# B&R Automation Studio project condmon
Automation Studio 4.6.3.55 SP

## Configuration X20CP3585

CPU X20CP3585, AutomationRuntime B4.62, Build 4.1.2, Safety 0.0, Vc 

### Task classes (Cpu.sw)
```
Cyclic#1 (cycle 1000 us, tolerance 1000 us):
  rdbuf <- rdbuf.prg
Binaries: udbdef, FWRules, TCData, iomap, ashwac, Role, sysconf, arconfig, asfw, User, ashwd, vccdt, vccbmp, Visu03, vccline, vcfile, arial, vctcal, vcrt, vcmgr, arsvcreg, vccstr, vcbclass, vccbtn, vcgclass, vcdsint, vcnet, vcchtml, Visu01, Visu, vcshared, vcclbox, vccddbox, vccscale, arialbd, vcxml, vccnum, vcpdvnc, vccalarm, vccurl, vccslider, vccbar, vcctext, vccpiech, vcpdsw, vcfntttf, vccovl, vccshape, vcalarm, vcpkat, Visu02, vcctrend, vccpopup, vcdsloc, vcchspot, vcpfx20, Config, Config_2, Config_1
Libraries: operator, runtime, astime, AsIecCon, AsIOVib, AsFltGen, brsystem, sys_lib, DataObj, asstring, standard, vcresman, asbrstr, ashw, MpAlarmX, MpFile, MpBase, AsSem, MpWebXs
```

### Hardware
```
X20BM31 : X20BM31 v1.0.0.1  [X2X1 -> X20CP3585.IF6]
X20CM4810 : X20CM4810 v1.4.4.0  [SS1 -> X20TB12.SS; SL -> X20BM31.SL1]
  Supervision = off
  Current01 = on
  FrequencyBandEnable01 = off
  FrequencyBandEnable02 = off
  FrequencyBandEnable03 = off
  FrequencyBandEnable09 = off
  FrequencyBandEnable10 = off
  FrequencyBandEnable11 = off
  FrequencyBandEnable17 = off
  FrequencyBandEnable18 = off
  FrequencyBandEnable19 = off
  FrequencyBandEnable25 = off
  FrequencyBandEnable26 = off
  FrequencyBandEnable27 = off
X20CP3585 : X20CP3585 v1.5.0.0
  Connector IF2:
    ActivateDevice = 1
    HostName = conmon
    Mode = Manual
    InternetAddress = 192.168.0.34
    SubnetMask = 255.255.255.0
  Connector IF6:
    CycleTime = 1000
    Stations = 16
    AsyncPayload = 160
    OutputJustInTime = off
  ConfigurationID = firstStart_X20CP3585
  Cyclic1Duration = 1000
  Cyclic1Tolerance = 1000
  FileDevice1
  FileDeviceName1 = HD
  FileDevicePath1 = F:\
  FtpUser1
  FtpUsername1 = user
  FtpUserPassword1 = IKmmIU0UA42VIUZbb7SMTTmDelvdeU0oRhYqfrVB1tM=
  FtpUserSalt1 = 73ZO5cbR
  FTPAccessRight1 = 0
X20TB12 : X20TB12 v1.0.0.0
```

### IoMap.iom - X20CP3585/IoMap.iom
```iecst
VAR_CONFIG
	::rdbuf:fb.ioMapping.RequestBufferLock01 AT %QX."X20CM4810".RequestBufferLock01;
	::rdbuf:fb.ioMapping.BufferLockValid01 AT %IX."X20CM4810".BufferLockValid01;
	::rdbuf:fb.ioMapping.BufferInputSequence01 AT %IB."X20CM4810".BufferInputSequence01;
	::rdbuf:fb.ioMapping.BufferRxByte01 AT %IB."X20CM4810".BufferRxByte01;
	::rdbuf:fb.ioMapping.BufferRxByte02 AT %IB."X20CM4810".BufferRxByte02;
	::rdbuf:fb.ioMapping.BufferRxByte03 AT %IB."X20CM4810".BufferRxByte03;
	::rdbuf:fb.ioMapping.BufferRxByte04 AT %IB."X20CM4810".BufferRxByte04;
	::rdbuf:fb.ioMapping.BufferRxByte05 AT %IB."X20CM4810".BufferRxByte05;
	::rdbuf:fb.ioMapping.BufferOutputSequence01 AT %QB."X20CM4810".BufferOutputSequence01;
	::rdbuf:fb.ioMapping.BufferTxByte01 AT %QB."X20CM4810".BufferTxByte01;
	::rdbuf:fb.ioMapping.BufferTxByte02 AT %QB."X20CM4810".BufferTxByte02;
	::rdbuf:fb.ioMapping.BufferTxByte03 AT %QB."X20CM4810".BufferTxByte03;
	::rdbuf:fb.ioMapping.BufferTxByte03 AT %QB."X20CM4810".BufferTxByte04;
END_VAR
```

## Logical view

Binary libraries used (declarations not repeated): operator, runtime, astime, AsIecCon, AsIOVib, AsFltGen, brsystem, sys_lib, DataObj, asstring, standard

### Global.typ - Globale Datentypen
```iecst
TYPE
	CM4810_Data : 	STRUCT
		xAxis : ARRAY[0..8191]OF REAL;
		yAxis : ARRAY[0..8191]OF REAL;
	END_STRUCT;
END_TYPE
```


### Program Logical/rdbuf (IEC)

#### Variables.var
```iecst
VAR
	fb : vbioCtrlCM4810Ex1;
	bufferUploadDuration : TIME;
	cmdUploadBuffer : USINT;
	cycleCounter : UDINT;
	step : UINT;
	rtinfo : RTInfo;
	moduleData : CM4810_Data; (*allgemeine Parameterstruktur*)
END_VAR
```

#### Main.st
```iecst
PROGRAM _INIT
	fb.paramMain.pModulePath := ADR('IF6.ST1');
	fb.paramMain.sensitivitySensor01 := 100;
	fb.paramMain.sensitivitySensor02 := 100;
	fb.paramMain.sensitivitySensor03 := 100;
	fb.paramMain.sensitivitySensor04 := 100;

	fb.paramBufferUpload.moduleBuffer := 9; (* Buffer: Rohsignal Beschleunigung Kanal 1 *)
	fb.paramBufferUpload.nrArrayElements:= SIZEOF(moduleData.xAxis)/SIZEOF(moduleData.xAxis[0]);
	fb.paramBufferUpload.pArrayXaxis:= ADR(moduleData.xAxis);
	fb.paramBufferUpload.pArrayYaxis:= ADR(moduleData.yAxis);
	fb.enable := 1;

	rtinfo.enable := 1;
	rtinfo();
	step := 0;

END_PROGRAM

PROGRAM _CYCLIC
	CASE( step) OF
		0:
		(* clear requests *)
		fb.requestBufferLock := 0;
		fb.uploadBuffer := 0;
		IF( fb.initDone AND fb.moduleCfgUploadDone )THEN
			step := 100;
		END_IF

		(* wait for command *)
		100:
		IF( cmdUploadBuffer = 1 )THEN
			cmdUploadBuffer := 2; (* busy *)
			step := 110;
		END_IF

		110:
		(* wait until buffer is locked *)
		fb.requestBufferLock := 1;  (* request for locking buffer *)
		IF( fb.bufferLockValid )THEN
			cycleCounter := 0;
			fb.uploadBuffer := 1;
			step := 120;
		END_IF

		120:
		cycleCounter := cycleCounter + 1 ;
		(* wait until buffer is uploaded *)
		IF( fb.bufferUploadDone )THEN
			(* do something with data *)
			fb.requestBufferLock := 0;  (* clear requests *)
			fb.uploadBuffer := 0;
			cmdUploadBuffer := 0; (* ready *)
			step := 100;
			bufferUploadDuration := (cycleCounter * rtinfo.cycle_time) / 1000;
		END_IF

	END_CASE
	fb();

END_PROGRAM

PROGRAM _EXIT
	(* Insert code here *)

END_PROGRAM
```

Listed in the project but not available here: Logical/Global.var
